PROGRAM MAIN
VAR
END_VAR

(*Include different program calls here*)

PRG_Example();


//Do Not Remove this
// Run the Diagnostics PRG
DIAGNOSTICS();

END_PROGRAM

(* stored: Version 1.1.0.1, ProductVersion 3.1.4022.16
   POU MAIN: Id {1ace9613-479b-4efe-9830-c468b81e6ab0}, SpecialFunc None *)
